ORGANIZATION_BLOCK "EnS_StartupOB"
TITLE = Startup OB
{ S7_Optimized_Access := 'TRUE' }
AUTHOR : Siemens
FAMILY : EnS
VERSION : 1.0
//Startup OB

BEGIN
	//FC for startup OB
	"EnS_StartupFC"();

END_ORGANIZATION_BLOCK

